TYPE ST_MESSAGEHEADER :
STRUCT
	CREATIONDATE	:STRING;
	CREATIONTIME	:STRING;
	MESSAGETYPE		:STRING;
	TESTINDICATOR	:STRING;
	SENDERSYSTEM	:STRING;
	RECEIVERSYSTEM	:STRING;
	REFERENCEID		:STRING;
	SOURCEID		:STRING;
END_STRUCT
END_TYPE

(* stored: Version 1.1.0.1, ProductVersion 3.1.4024.13
   DUT ST_MESSAGEHEADER: Id {c1e16df8-ada8-47e3-9cd1-5b11623c9c0d} *)
